Omron CX-Programmer project 新工程 (CX-Programmer 9.61)

# PLC 新PLC1: CP1E N30

## Global symbols (name address type ; comment)
0.06 BOOL  ; 退钱
100.00 BOOL  ; 口香糖指示灯
100.01 BOOL  ; 饮料指示灯
100.02 BOOL  ; 口香糖闪烁控制
100.03 BOOL  ; 饮料闪烁控制
100.05 BOOL  ; 退钱指示灯
D100 CHANNEL  ; 1元硬币
D101 CHANNEL  ; 5元硬币
D102 CHANNEL  ; 10元硬币
D103 CHANNEL  ; 口香糖指示灯
D104 CHANNEL  ; 口香糖
D105 CHANNEL  ; 饮料
D106 CHANNEL  ; 饮料指示灯
D120 CHANNEL  ; 总计硬币

## Program 新程序1 (cyclic task 0)

### Section 段1

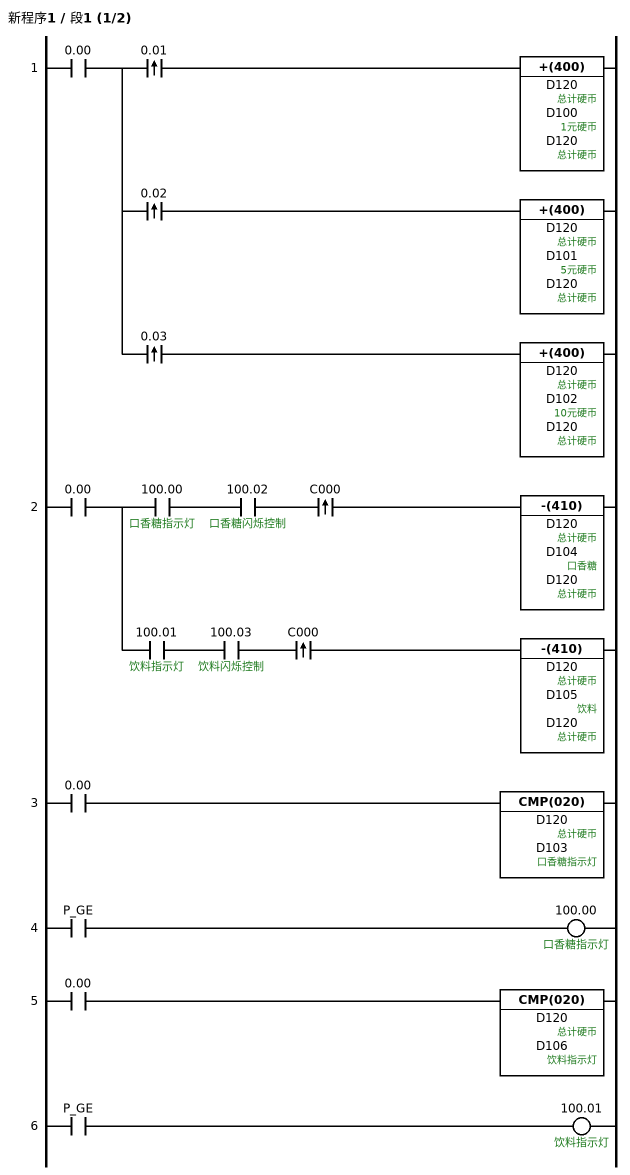
; rung 1
LD 0.00
OUT TR0
@AND 0.01
+(400) D120 D100 D120  ; 总计硬币, 1元硬币
LD TR0
@AND 0.02
+(400) D120 D101 D120  ; 总计硬币, 5元硬币
LD TR0
@AND 0.03
+(400) D120 D102 D120  ; 总计硬币, 10元硬币
; rung 2
LD 0.00
OUT TR0
AND 100.00  ; 口香糖指示灯
AND 100.02  ; 口香糖闪烁控制
@AND C000
-(410) D120 D104 D120  ; 总计硬币, 口香糖
LD TR0
AND 100.01  ; 饮料指示灯
AND 100.03  ; 饮料闪烁控制
@AND C000
-(410) D120 D105 D120  ; 总计硬币, 饮料
; rung 3
LD 0.00
CMP(020) D120 D103  ; 总计硬币, 口香糖指示灯
; rung 4
LD P_GE
OUT 100.00  ; 口香糖指示灯
; rung 5
LD 0.00
CMP(020) D120 D106  ; 总计硬币, 饮料指示灯
; rung 6
LD P_GE
OUT 100.01  ; 饮料指示灯

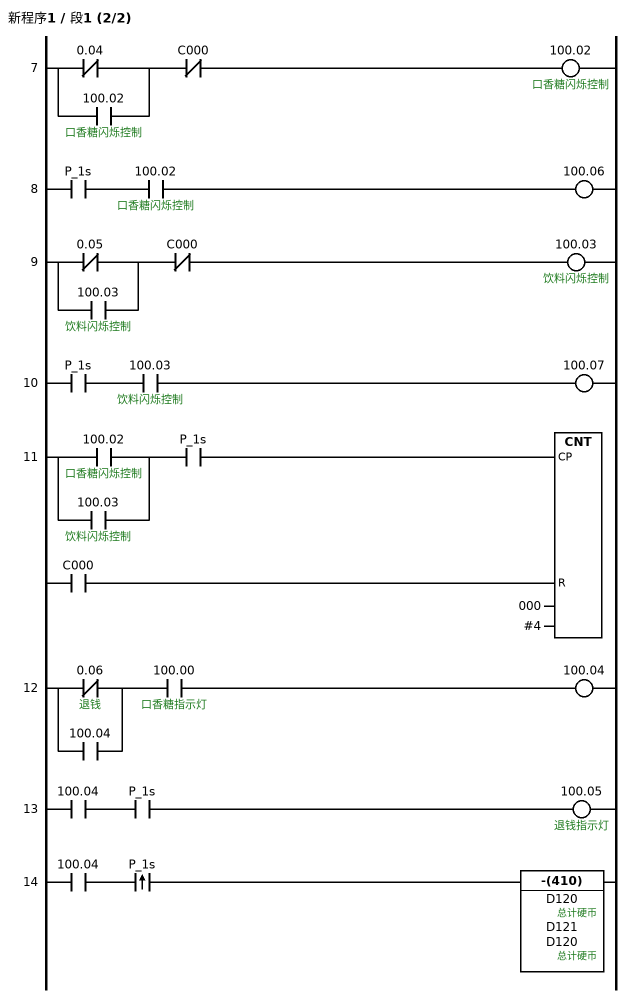
; rung 7
LDNOT 0.04
OR 100.02  ; 口香糖闪烁控制
ANDNOT C000
OUT 100.02  ; 口香糖闪烁控制
; rung 8
LD P_1s
AND 100.02  ; 口香糖闪烁控制
OUT 100.06
; rung 9
LDNOT 0.05
OR 100.03  ; 饮料闪烁控制
ANDNOT C000
OUT 100.03  ; 饮料闪烁控制
; rung 10
LD P_1s
AND 100.03  ; 饮料闪烁控制
OUT 100.07
; rung 11
LD 100.02  ; 口香糖闪烁控制
OR 100.03  ; 饮料闪烁控制
AND P_1s
LD C000
CNT 000 #4
; rung 12
LDNOT 0.06  ; 退钱
OR 100.04
AND 100.00  ; 口香糖指示灯
OUT 100.04
; rung 13
LD 100.04
AND P_1s
OUT 100.05  ; 退钱指示灯
; rung 14
LD 100.04
@AND P_1s
-(410) D120 D121 D120  ; 总计硬币
; rung 15
END(001)

### Section END
; rung 0
END(001)